// TIA Portal V19 export
DATA_BLOCK "EnS_Calc_InfeedPAC3200"   // DB22
TITLE = Instance DB of calculation function
// Instance DB of calculation function
// stored: InstanceOfName EnS_CalcEnergyData, InstanceOfType FB
"EnS_CalcEnergyData"
   // VAR_INPUT
   //    power { ExternalAccessible := 'False'; ExternalVisible := 'False'; ExternalWritable := 'False'} : "EnS_typeAnalogValue";
   //    energy { ExternalAccessible := 'False'; ExternalVisible := 'False'; ExternalWritable := 'False'} : "EnS_typeEnergyCounter";
   // END_VAR
   // VAR_OUTPUT
   //    energyBasic { ExternalAccessible := 'False'; ExternalVisible := 'False'; ExternalWritable := 'False'} : "EnS_typeEnergyBasic";
   //    error { ExternalAccessible := 'False'; ExternalVisible := 'False'; ExternalWritable := 'False'} : Bool;
   //    status { ExternalAccessible := 'False'; ExternalVisible := 'False'; ExternalWritable := 'False'} : Word;
   // END_VAR
   // VAR_IN_OUT
   //    orgData : "EnS_typeOrgData";
   //    syncData : "EnS_typeSync";
   //    energyMeta : "EnS_typeEnergyMeta";
   // END_VAR
   // VAR
   //    sr64_EnergyNormValueOld { ExternalAccessible := 'False'; ExternalVisible := 'False'; ExternalWritable := 'False'} : LReal;
   //    sr64_ActEnergyNormValueOld { ExternalAccessible := 'False'; ExternalVisible := 'False'; ExternalWritable := 'False'} : LReal;
   //    sr64_ActEnergy { ExternalAccessible := 'False'; ExternalVisible := 'False'; ExternalWritable := 'False'} : LReal;
   //    sr64_EnergyPwr { ExternalAccessible := 'False'; ExternalVisible := 'False'; ExternalWritable := 'False'} : LReal;
   //    sr64_EnergyPwrOld { ExternalAccessible := 'False'; ExternalVisible := 'False'; ExternalWritable := 'False'} : LReal;
   //    sr32_ActPower { ExternalAccessible := 'False'; ExternalVisible := 'False'; ExternalWritable := 'False'} : Real;
   //    sr32_SyncPeriod { ExternalAccessible := 'False'; ExternalVisible := 'False'; ExternalWritable := 'False'} : Real;
   //    su16_OverflowEnergyCounter { ExternalAccessible := 'False'; ExternalVisible := 'False'; ExternalWritable := 'False'} : UInt;
   //    su16_UnderflowEnergyCounter { ExternalAccessible := 'False'; ExternalVisible := 'False'; ExternalWritable := 'False'} : UInt;
   //    su32_AcqTime { ExternalAccessible := 'False'; ExternalVisible := 'False'; ExternalWritable := 'False'} : UDInt;
   //    sb16_StatusEnergy { ExternalAccessible := 'False'; ExternalVisible := 'False'; ExternalWritable := 'False'} : Word;
   //    sb16_StatusPower { ExternalAccessible := 'False'; ExternalVisible := 'False'; ExternalWritable := 'False'} : Word;
   //    sb16_StatusActEnergy { ExternalAccessible := 'False'; ExternalVisible := 'False'; ExternalWritable := 'False'} : Word;
   //    sb16_StatusActPower { ExternalAccessible := 'False'; ExternalVisible := 'False'; ExternalWritable := 'False'} : Word;
   //    sb16_StatusOld { ExternalAccessible := 'False'; ExternalVisible := 'False'; ExternalWritable := 'False'} : Word;
   //    sb16_StatusEnergyOld { ExternalAccessible := 'False'; ExternalVisible := 'False'; ExternalWritable := 'False'} : Word;
   //    sb16_StatusPowerOld { ExternalAccessible := 'False'; ExternalVisible := 'False'; ExternalWritable := 'False'} : Word;
   //    sb16_StatusSync { ExternalAccessible := 'False'; ExternalVisible := 'False'; ExternalWritable := 'False'} : Word;
   //    sb16_StatusParam { ExternalAccessible := 'False'; ExternalVisible := 'False'; ExternalWritable := 'False'} : Word;
   //    sbo_SyncPulseOld { ExternalAccessible := 'False'; ExternalVisible := 'False'; ExternalWritable := 'False'} : Bool;
   //    sbo_Sync { ExternalAccessible := 'False'; ExternalVisible := 'False'; ExternalWritable := 'False'} : Bool;
   //    sbo_ValueChanged { ExternalAccessible := 'False'; ExternalVisible := 'False'; ExternalWritable := 'False'} : Bool;
   //    sbo_Init { ExternalAccessible := 'False'; ExternalVisible := 'False'; ExternalWritable := 'False'} : Bool;
   // END_VAR
BEGIN
END_DATA_BLOCK
